# EPICS StreamDevice protocol: MKS660.proto
Terminator = CR LF;
LockTimeout = 10000;
ReplyTimeout = 1000;
ReadTimeout = 500;
WriteTimeout = 1000;

#This command is used to read the pressures
ReadPressure	{
   out "R5"; in "P%f"
}
